{attribute addProperty BoxType "EL6201-0000-0017"}
{attribute addProperty Id "Slave_29A_DO0BIT10.125225Slave_29A_DO1BIT10.125226Slave_29A_DO2BIT10.125227Slave_29A_DO3BIT10.125228Slave_29B_DO0BIT10.125229Slave_29B_DO1BIT10.125230Slave_29B_DO2BIT10.125231Slave_29B_DO3BIT10.125232"}
{attribute addProperty CRC "1651599084"}
{attribute addProperty SizeInBites "8"}
{attribute addProperty SizeInBytes "1"}
TYPE Slave_29_Outputs_627166EC :
STRUCT
	{attribute addProperty Name "Slave_29A_DO0"}
	Slave_29A_DO0 : BIT;
	{attribute addProperty Name "Slave_29A_DO1"}
	Slave_29A_DO1 : BIT;
	{attribute addProperty Name "Slave_29A_DO2"}
	Slave_29A_DO2 : BIT;
	{attribute addProperty Name "Slave_29A_DO3"}
	Slave_29A_DO3 : BIT;
	{attribute addProperty Name "Slave_29B_DO0"}
	Slave_29B_DO0 : BIT;
	{attribute addProperty Name "Slave_29B_DO1"}
	Slave_29B_DO1 : BIT;
	{attribute addProperty Name "Slave_29B_DO2"}
	Slave_29B_DO2 : BIT;
	{attribute addProperty Name "Slave_29B_DO3"}
	Slave_29B_DO3 : BIT;
END_STRUCT
END_TYPE

(* stored: Version 1.2.0.0, ProductVersion 3.1.4024.9
   DUT Slave_29_Outputs_627166EC: Id {0b0ce1a2-9440-490d-bb55-8894418f9c99} *)
